FUNCTION_BLOCK FB_HwModule
VAR_INPUT
END_VAR
VAR_OUTPUT
END_VAR
VAR
	stHardwareId : ST_HardwareId;
	bBusy : BOOL;
	bError : BOOL;
	stError : ST_Error;
END_VAR

METHOD M_GetHwInfo : ST_HardwareInfo
VAR_INPUT
END_VAR

VAR
	nHwId : UDINT;
END_VAR
nHwId := SHL(UINT_TO_UDINT(stHardwareId.eGroup),16);
nHwId := nHwId OR (SHL(UINT_TO_UDINT(stHardwareId.nParentItem),8));
nHwId := nHwId OR stHardwareId.nItem;
M_GetHwInfo.nHwId := nHwId;
END_METHOD

METHOD M_Reset
VAR_INPUT
END_VAR
END_METHOD

PROPERTY P_bBusy : BOOL
GET
P_bBusy := bBusy;
END_GET
END_PROPERTY

PROPERTY P_bError : BOOL
GET
P_bError := bError;
END_GET
END_PROPERTY

PROPERTY P_eHardwareGrp : E_HardwareGrp
GET
P_eHardwareGrp := stHardwareId.eGroup;
END_GET
END_PROPERTY

PROPERTY P_stError : ST_Error
GET
P_stError := stError;
END_GET
END_PROPERTY

PROPERTY P_stHardwareId : ST_HardwareId
GET
P_stHardwareId := stHardwareId;
END_GET
SET
stHardwareId := P_stHardwareId;
END_SET
END_PROPERTY

END_FUNCTION_BLOCK

(* stored: Version 1.1.0.1, ProductVersion 3.1.4022.10
   POU FB_HwModule: Id {151b4dca-e858-44b2-a722-4a4d4931cf5e}, SpecialFunc None
   Method M_GetHwInfo: Id {aacf537f-c2a3-45d5-8d0c-38e3e45704dd}
   Method M_Reset: Id {87b8d77e-bb50-4562-8dee-a6cc9e705e21}
   Property P_bBusy: Id {16a8a61d-c097-4af6-bbf3-01065605f1bd}
   Get Get: Id {6d716fdf-22a4-4fdb-b0b9-fb5ad40fa00f}
   Property P_bError: Id {3aeb50aa-f1fc-494f-9cef-837f51f4a155}
   Get Get: Id {3f3cf82c-8176-484c-b44e-102e63603a2a}
   Property P_eHardwareGrp: Id {479e2b5d-f5d6-41fb-a80c-f1a55e50c66b}
   Get Get: Id {3173f508-aa30-4293-8813-b8c03b746ee1}
   Property P_stError: Id {39aad715-953d-46c0-b66f-646dd2200afe}
   Get Get: Id {f168966a-20d4-4a73-8aa5-dedab4c6821c}
   Property P_stHardwareId: Id {6e4629b3-db27-476c-bb33-592e266fe2ac}
   Get Get: Id {bb5a3a70-e773-49cb-ae5c-34dc4d9a0a09}
   Set Set: Id {a9ab0989-605e-44bb-bc2d-b5fd9d652b94} *)
